// TIA Portal V18 export
FUNCTION_BLOCK "Main_Safety_RTG1"   // FB1, F_FBD
{ S7_Optimized_Access := 'TRUE' }
// stored: AutoNumber false
BEGIN
END_FUNCTION_BLOCK
